Fanuc KAREL source: kb00068.KL

-- PROVISIONAL review KL for V1013-1; original PC SHA256 2d42d211f1456c055d58f1e59ec10c65362e00cc482d39a2e9c510f3c5fcfa6f
-- Incomplete behavior may be omitted. Consult companion uncertainty JSON. Do not deploy.
PROGRAM KB00068
%NOLOCKGROUP
BEGIN
  -- UNRESOLVED_PC offsets 5-14; opcodes 3F,75
  -- UNRESOLVED_PC offsets 19-26; opcodes 9D,23
  -- UNRESOLVED_PC offsets 31-49; opcodes 27,22,2A,22,31
  -- UNRESOLVED_PC offsets 54-58; opcodes 7F
END KB00068
